Yaskawa INFORM job: R1-S1-NONCOORD.JBI

/JOB
//NAME R1-S1-NONCOORD
//POS
///NPOS 4,0,4,0,0,0
///TOOL 0
///POSTYPE PULSE
///PULSE
C00000=-5697,-22758,-19385,-13694,-18452,6429
C00001=-6744,-46438,-34826,-14046,-21223,6588
C00002=-6744,-46438,-34826,-14046,-21223,6588
C00003=-5766,-24566,-20667,-13744,-18600,6452
EC00000=-14293,247808
EC00001=-14293,247808
EC00002=-28898,221232
EC00003=-28898,221232
//INST
///DATE 2023/01/18 18:15
///ATTR SC,RW
///GROUP1 RB1,ST1
NOP
MOVJ C00000 EC00000 VJ=0.78
MOVJ C00001 EC00001 VJ=0.78
MOVJ C00002 EC00002 VJ=0.78
MOVL C00003 EC00003 V=11.0
END
